// TIA Portal V18 export
// export: Created 2023-08-17T07:23:58.0636782Z, ExportSetting WithDefaults, DisplayName Totally Integrated Automation Portal, DisplayVersion V18 Update 2, DisplayName TIA Portal Openness, DisplayVersion V18 Update 2, DisplayName TIA Portal Version Control Interface, DisplayVersion V18, DisplayName SINAMICS Startdrive Advanced, DisplayVersion V18, DisplayName SINAMICS Startdrive G130, G150, S120, S150, SINAMICS MV, S210, DisplayVersion V18, DisplayName SINAMICS Startdrive G110M, G120, G120C, G120D, G120P, G115D, DisplayVersion V18, DisplayName STEP 7 Professional, DisplayVersion V18 Update 2, DisplayName STEP 7 Safety, DisplayVersion V18, DisplayName WinCC Advanced / Unified PC, DisplayVersion V18 Update 2
ORGANIZATION_BLOCK "Drives"   // OB124, LAD, ProgramCycle
TITLE = "Main Program Sweep (Cycle)"
{ S7_Optimized_Access := 'TRUE' }
VERSION : 0.1
// stored: AutoNumber true, IsIECCheckEnabled false, SetENOAutomatically false
   VAR_INPUT
      Initial_Call : Bool;   // Initial call of this OB
      Remanence : Bool;   // =True, if remanent data are available
   END_VAR
BEGIN

REGION Network 1
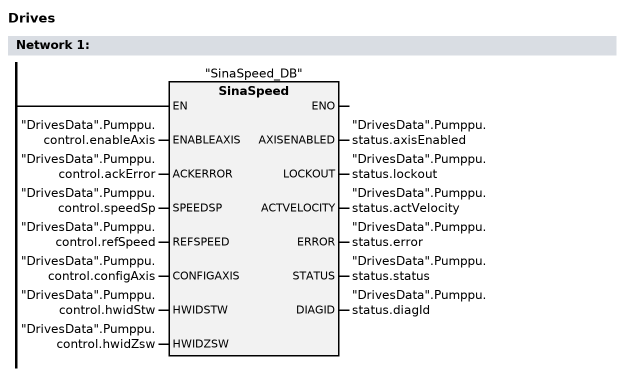
   RUNG wire#powerrail
      "SinaSpeed_DB".SinaSpeed(EnableAxis := "DrivesData".Pumppu.control.enableAxis, AckError := "DrivesData".Pumppu.control.ackError, SpeedSp := "DrivesData".Pumppu.control.speedSp, RefSpeed := "DrivesData".Pumppu.control.refSpeed, ConfigAxis := "DrivesData".Pumppu.control.configAxis, HWIDSTW := "DrivesData".Pumppu.control.hwidStw, HWIDZSW := "DrivesData".Pumppu.control.hwidZsw, AxisEnabled => "DrivesData".Pumppu.status.axisEnabled, Lockout => "DrivesData".Pumppu.status.lockout, ActVelocity => "DrivesData".Pumppu.status.actVelocity, Error => "DrivesData".Pumppu.status.error, Status => "DrivesData".Pumppu.status.status, DiagId => "DrivesData".Pumppu.status.diagId)
   END_RUNG
   // the same network as SCL:
   "SinaSpeed_DB"(EnableAxis := "DrivesData".Pumppu.control.enableAxis,   // SinaSpeed
                  AckError := "DrivesData".Pumppu.control.ackError,
                  SpeedSp := "DrivesData".Pumppu.control.speedSp,
                  RefSpeed := "DrivesData".Pumppu.control.refSpeed,
                  ConfigAxis := "DrivesData".Pumppu.control.configAxis,
                  HWIDSTW := "DrivesData".Pumppu.control.hwidStw,
                  HWIDZSW := "DrivesData".Pumppu.control.hwidZsw,
                  AxisEnabled => "DrivesData".Pumppu.status.axisEnabled,
                  Lockout => "DrivesData".Pumppu.status.lockout,
                  ActVelocity => "DrivesData".Pumppu.status.actVelocity,
                  Error => "DrivesData".Pumppu.status.error,
                  Status => "DrivesData".Pumppu.status.status,
                  DiagId => "DrivesData".Pumppu.status.diagId);
END_REGION
END_ORGANIZATION_BLOCK
